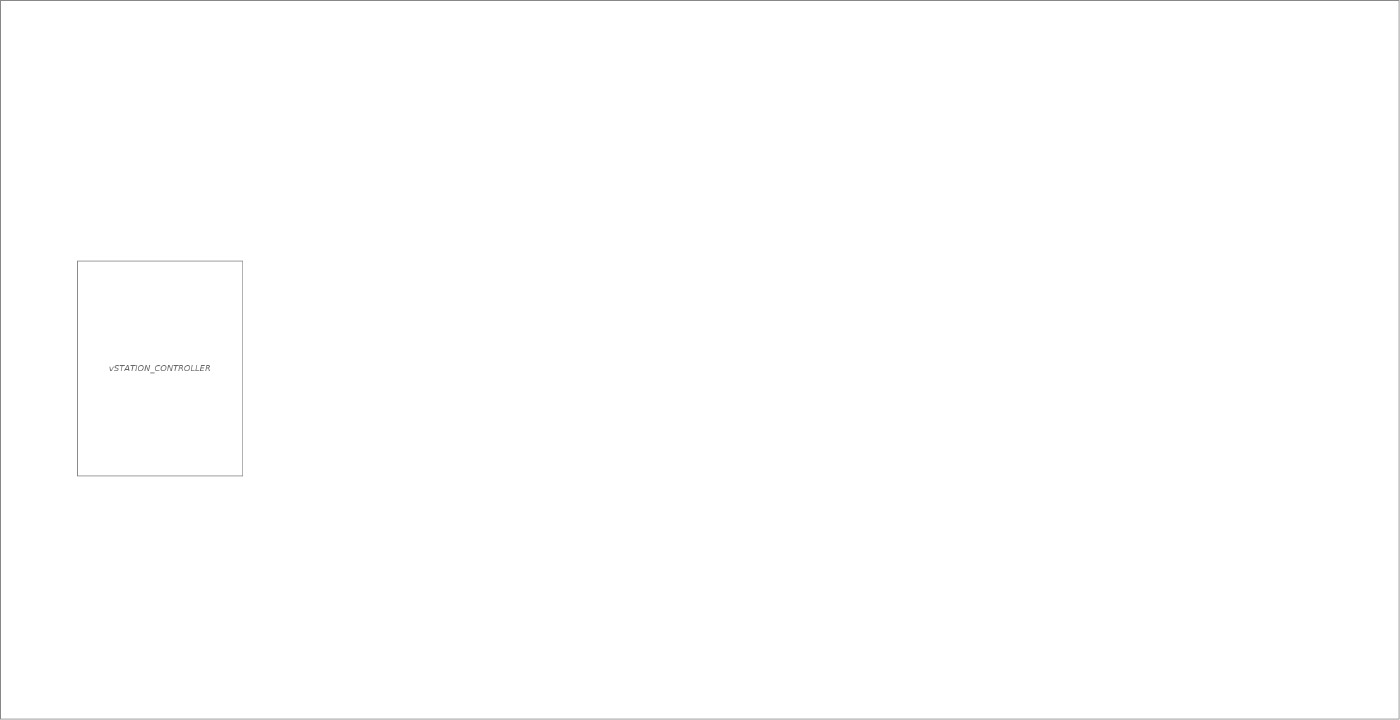
VISUALIZATION vMACHINE  // 1690x870
    Frame (93,315 200x260)
        shows vSTATION_CONTROLLER(vSTATION := fbFEEDER)
END_VISUALIZATION

(* stored: Version 1.1.0.1, ProductVersion 3.1.4024.12
   Visu vMACHINE: Id {3deaac7f-3d0e-48ef-a7db-42e8b819f786} *)
